{attribute 'GeneratedUsingTerminal: EL9560-0000-0016'}
{attribute addProperty BoxType "EL9560-0000-0016"}
{attribute addProperty Id "EtcSlaveTerminalBaseStatus_UsAT %I*Status_Us_449D6AB51Status_UoAT %I*Status_Uo_449D6AB51WcStateAT %I*WcState_9091E0EB2InfoDataAT %I*InfoData_6F19DB2B2"}
{attribute addProperty CRC "3139611612"}
{attribute addProperty Size "6"}
TYPE EL9560_BB22ABDC EXTENDS EtcSlaveTerminalBase :
STRUCT
	{attribute addProperty Name "Status_Us"}
	Status_Us : Status_Us_449D6AB5;
	{attribute addProperty Name "Status_Uo"}
	Status_Uo : Status_Uo_449D6AB5;
	{attribute addProperty Name "WcState"}
	WcState : WcState_9091E0EB;
	{attribute addProperty Name "InfoData"}
	InfoData : InfoData_6F19DB2B;
END_STRUCT
END_TYPE

(* stored: Version 1.2.0.0, ProductVersion 3.1.4024.9
   DUT EL9560_BB22ABDC: Id {61c195ec-3e45-46fd-9831-1fb7f075ce1d} *)
